// TIA Portal V17 export
// export: Created 2023-02-26T22:53:29.6504216Z, ExportSetting WithDefaults, DisplayName Totally Integrated Automation Portal, DisplayVersion V17, DisplayName TIA Portal Openness, DisplayVersion V17, DisplayName TIA Portal Version Control Interface, DisplayVersion V17, DisplayName TIA Portal Test Suite Advanced, DisplayVersion V17, DisplayName STEP 7 Professional, DisplayVersion V17, DisplayName SIMATIC Energy Suite, DisplayVersion V17, DisplayName STEP 7 Safety, DisplayVersion V17, DisplayName WinCC Professional, DisplayVersion V17
FUNCTION "ERR_LostPackages" : Void   // FC12, LAD
{ S7_Optimized_Access := 'TRUE' }
VERSION : 0.1
// stored: AutoNumber true, IsIECCheckEnabled false, SetENOAutomatically false, UDAEnableTagReadback false
   VAR_INPUT
      StartLine : Bool;
      StopLine : Bool;
      AutoMode : Bool;
      ResetButton : Bool;
      FirstScan : Bool;
   END_VAR
   VAR_OUTPUT
      Error : "stt_LostPackageError";
   END_VAR
BEGIN

REGION Network 1: Call: LostPackage - error 1
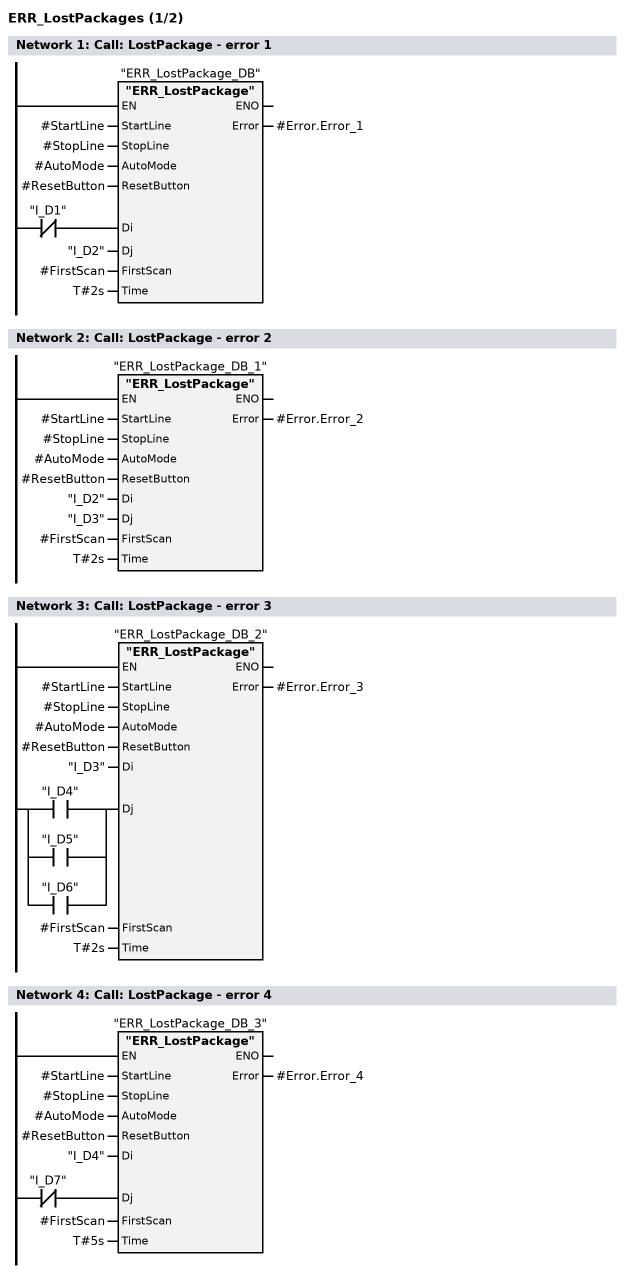
   RUNG wire#powerrail
      "ERR_LostPackage_DB"(Di := wire#w1, StartLine := #StartLine, StopLine := #StopLine, AutoMode := #AutoMode, ResetButton := #ResetButton, Dj := "I_D2", FirstScan := #FirstScan, "Time" := T#2s, Error => #Error.Error_1)
   END_RUNG
   RUNG wire#powerrail
      I_Contact( "I_D1" )
   END_RUNG wire#w1
   // the same network as SCL:
   "ERR_LostPackage_DB"(StartLine := #StartLine,   // "ERR_LostPackage"
                        StopLine := #StopLine,
                        AutoMode := #AutoMode,
                        ResetButton := #ResetButton,
                        Di := NOT "I_D1",
                        Dj := "I_D2",
                        FirstScan := #FirstScan,
                        "Time" := T#2s,
                        Error => #Error.Error_1);
END_REGION

REGION Network 2: Call: LostPackage - error 2
   RUNG wire#powerrail
      "ERR_LostPackage_DB_1"(StartLine := #StartLine, StopLine := #StopLine, AutoMode := #AutoMode, ResetButton := #ResetButton, Di := "I_D2", Dj := "I_D3", FirstScan := #FirstScan, "Time" := T#2s, Error => #Error.Error_2)
   END_RUNG
   // the same network as SCL:
   "ERR_LostPackage_DB_1"(StartLine := #StartLine,   // "ERR_LostPackage"
                          StopLine := #StopLine,
                          AutoMode := #AutoMode,
                          ResetButton := #ResetButton,
                          Di := "I_D2",
                          Dj := "I_D3",
                          FirstScan := #FirstScan,
                          "Time" := T#2s,
                          Error => #Error.Error_2);
END_REGION

REGION Network 3: Call: LostPackage - error 3
   RUNG wire#powerrail
      "ERR_LostPackage_DB_2"(Dj := wire#w1, StartLine := #StartLine, StopLine := #StopLine, AutoMode := #AutoMode, ResetButton := #ResetButton, Di := "I_D3", FirstScan := #FirstScan, "Time" := T#2s, Error => #Error.Error_3)
   END_RUNG
   RUNG wire#powerrail
      Contact( "I_D4" )
   END_RUNG wire#w1
   RUNG wire#powerrail
      Contact( "I_D5" )
   END_RUNG wire#w1
   RUNG wire#powerrail
      Contact( "I_D6" )
   END_RUNG wire#w1
   // the same network as SCL:
   "ERR_LostPackage_DB_2"(StartLine := #StartLine,   // "ERR_LostPackage"
                          StopLine := #StopLine,
                          AutoMode := #AutoMode,
                          ResetButton := #ResetButton,
                          Di := "I_D3",
                          Dj := "I_D4" OR "I_D5" OR "I_D6",
                          FirstScan := #FirstScan,
                          "Time" := T#2s,
                          Error => #Error.Error_3);
END_REGION

REGION Network 4: Call: LostPackage - error 4
   RUNG wire#powerrail
      "ERR_LostPackage_DB_3"(Dj := wire#w1, StartLine := #StartLine, StopLine := #StopLine, AutoMode := #AutoMode, ResetButton := #ResetButton, Di := "I_D4", FirstScan := #FirstScan, "Time" := T#5s, Error => #Error.Error_4)
   END_RUNG
   RUNG wire#powerrail
      I_Contact( "I_D7" )
   END_RUNG wire#w1
   // the same network as SCL:
   "ERR_LostPackage_DB_3"(StartLine := #StartLine,   // "ERR_LostPackage"
                          StopLine := #StopLine,
                          AutoMode := #AutoMode,
                          ResetButton := #ResetButton,
                          Di := "I_D4",
                          Dj := NOT "I_D7",
                          FirstScan := #FirstScan,
                          "Time" := T#5s,
                          Error => #Error.Error_4);
END_REGION

REGION Network 5: Call: LostPackage - error 5
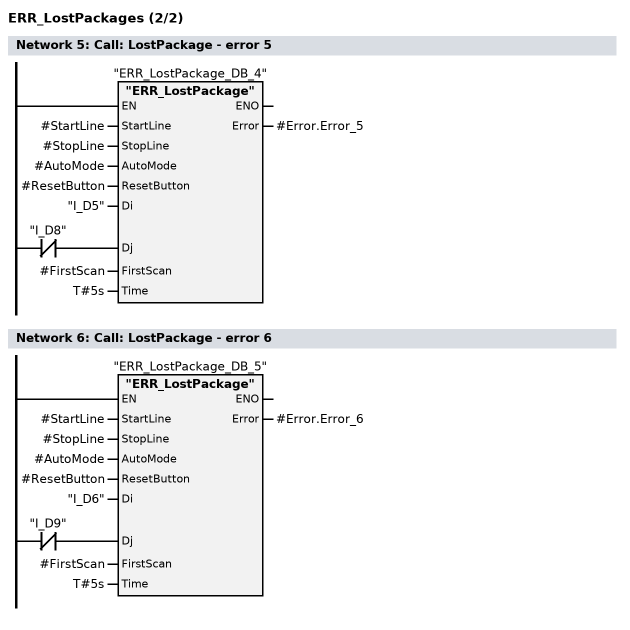
   RUNG wire#powerrail
      "ERR_LostPackage_DB_4"(Dj := wire#w1, StartLine := #StartLine, StopLine := #StopLine, AutoMode := #AutoMode, ResetButton := #ResetButton, Di := "I_D5", FirstScan := #FirstScan, "Time" := T#5s, Error => #Error.Error_5)
   END_RUNG
   RUNG wire#powerrail
      I_Contact( "I_D8" )
   END_RUNG wire#w1
   // the same network as SCL:
   "ERR_LostPackage_DB_4"(StartLine := #StartLine,   // "ERR_LostPackage"
                          StopLine := #StopLine,
                          AutoMode := #AutoMode,
                          ResetButton := #ResetButton,
                          Di := "I_D5",
                          Dj := NOT "I_D8",
                          FirstScan := #FirstScan,
                          "Time" := T#5s,
                          Error => #Error.Error_5);
END_REGION

REGION Network 6: Call: LostPackage - error 6
   RUNG wire#powerrail
      "ERR_LostPackage_DB_5"(Dj := wire#w1, StartLine := #StartLine, StopLine := #StopLine, AutoMode := #AutoMode, ResetButton := #ResetButton, Di := "I_D6", FirstScan := #FirstScan, "Time" := T#5s, Error => #Error.Error_6)
   END_RUNG
   RUNG wire#powerrail
      I_Contact( "I_D9" )
   END_RUNG wire#w1
   // the same network as SCL:
   "ERR_LostPackage_DB_5"(StartLine := #StartLine,   // "ERR_LostPackage"
                          StopLine := #StopLine,
                          AutoMode := #AutoMode,
                          ResetButton := #ResetButton,
                          Di := "I_D6",
                          Dj := NOT "I_D9",
                          FirstScan := #FirstScan,
                          "Time" := T#5s,
                          Error => #Error.Error_6);
END_REGION
END_FUNCTION
